ABB RobotStudio station: Romantici.rsstn

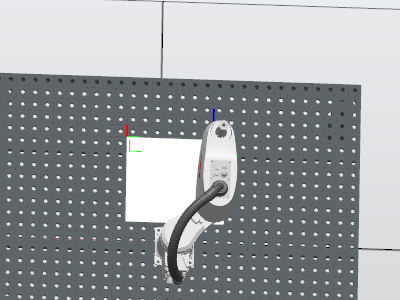
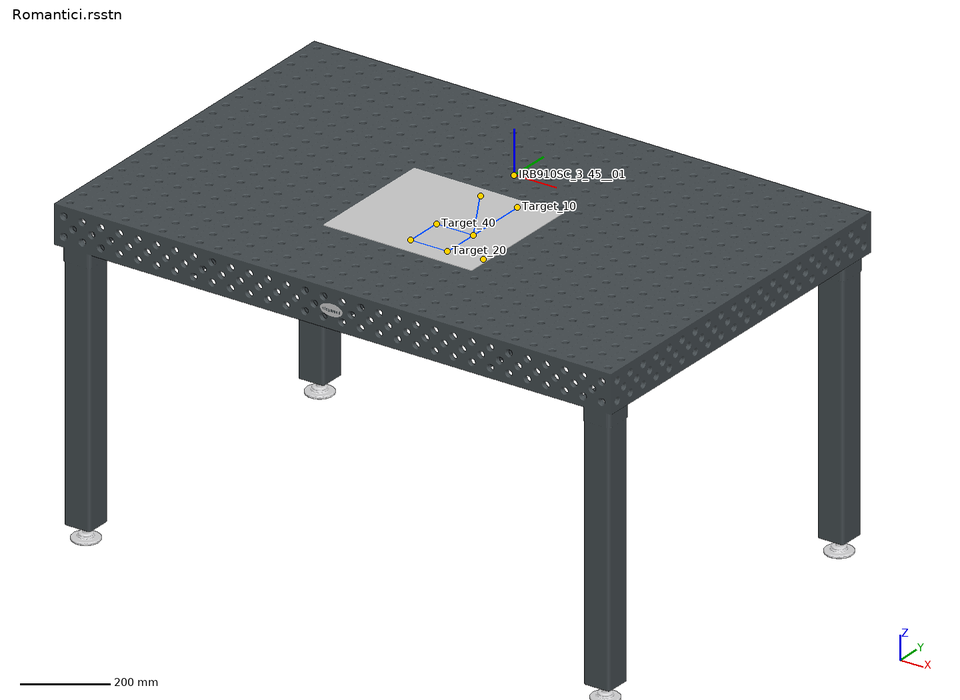
[picture v1: parts stored in the station drawn from their meshes, with robot base, taught points and paths (robot models come from the ABB library and are not in the file)]
Station Solution_1_Tutorial (saved by RobotStudio 22.3.10190.2)
Controller Controller3, task T_ROB1: task frame (RAPID world) sits at (0, 200, 830) mm, rotated rx 0 ry 0 rz -90 deg in the station
Controller Controller3
  mechanical unit ROB_1: IRB910SC_3_45__01, 4 joints, base frame (0, 0, 0) mm
Layout (positions relative to the parent item):
  - table [part] at (-200, -500, 830) mm
  - siegmund_1500_1000 [part], size 1500 x 1010.3 x 830 mm
  - IRB910SC_3_45__01 [mechanism, from Robots\IRB910SC_3_45__01.rslib] at (0, 200, 830) mm, rotated rx 0 ry 0 rz -90 deg; joint values [-2.1543, 2.1819, -0.0556, 0.0276] (rad or m)
  - PencilHolder [mechanism] at (-160, 60.29, 994.64) mm, rotated rx 180 ry 0 rz -90 deg
      TCP PencilHolder at (-72.46, -108.4, 17) mm, rotated rx 90 ry 0 rz 0 deg
      links: Assembly3
  - PAPER [part] at (-200, -250, 830) mm, size 400 x 350 x 2 mm
  - Rámec_1 [frame] at (0, 30, 162.64) mm, rotated rx 90 ry 0 rz -90 deg
Attachment: PencilHolder is attached to IRB910SC_3_45__01 / Link4
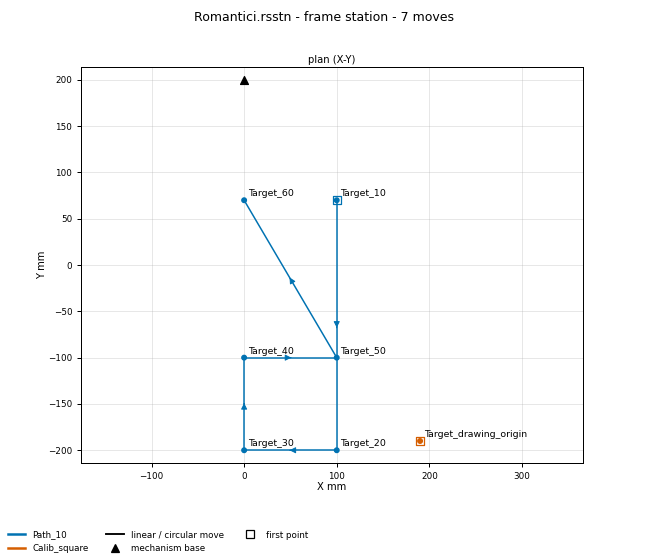
[picture p0: tool path of Romantici.rsstn in frame station, 7 of 7 moves have a stored position in this frame; points joined in program order, loops and branches not executed]
Targets, tools, work objects and paths stored in the station, written as RAPID:
! task T_ROB1
MODULE Module1
  PROC main()
  ENDPROC
ENDMODULE

! task T_ROB2
MODULE Module1
  PROC main()
  ENDPROC
ENDMODULE

! task T_ROB1
MODULE CalibData
  PERS tooldata PencilHolder:=[TRUE,[[0,30,162.643],[1,0,0,0]],[1,[0,0,1],[1,0,0,0],0,0,0]];
  PERS tooldata Pen_TCP:=[TRUE,[[110,0,140],[0.707106781,0,0.707106781,0]],[1,[10.7435139,0,140],[1,0,0,0],0,0,0]];
  TASK PERS wobjdata PAPER:=[FALSE,TRUE,"",[[100,200,0],[0,1,0,0]],[[0,0,0],[1,0,0,0]]];
ENDMODULE

! task T_ROB1
MODULE Module1
  CONST robtarget Target_10:=[[30,100,0],[1,0,0,0],[0,0,0,0],[9E+09,9E+09,9E+09,9E+09,9E+09,9E+09]];
  CONST robtarget Target_20:=[[300,100,0],[1,0,0,0],[0,0,0,0],[9E+09,9E+09,9E+09,9E+09,9E+09,9E+09]];
  CONST robtarget Target_30:=[[300,200,0],[1,0,0,0],[0,0,0,0],[9E+09,9E+09,9E+09,9E+09,9E+09,9E+09]];
  CONST robtarget Target_40:=[[200,200,0],[1,0,0,0],[0,0,0,0],[9E+09,9E+09,9E+09,9E+09,9E+09,9E+09]];
  CONST robtarget Target_50:=[[200,100,0],[1,0,0,0],[0,0,0,0],[9E+09,9E+09,9E+09,9E+09,9E+09,9E+09]];
  CONST robtarget Target_60:=[[30,200,0],[1,0,0,0],[0,0,0,0],[9E+09,9E+09,9E+09,9E+09,9E+09,9E+09]];
  CONST robtarget Target_corner:=[[350,0,-2],[1,0,0,0],[0,0,0,0],[9E+09,9E+09,9E+09,9E+09,9E+09,9E+09]];
  CONST robtarget Target_drawing_origin:=[[290,10,-2],[1,0,0,0],[0,0,0,0],[9E+09,9E+09,9E+09,9E+09,9E+09,9E+09]];
  CONST robtarget Target_opposite_corner:=[[100,390,-2],[1,0,0,0],[0,0,0,0],[9E+09,9E+09,9E+09,9E+09,9E+09,9E+09]];
  PROC Path_10()
    MoveL Target_10,v1000,z0,PencilHolder\WObj:=PAPER;
    MoveL Target_20,v1000,z0,PencilHolder\WObj:=PAPER;
    MoveL Target_30,v1000,z0,PencilHolder\WObj:=PAPER;
    MoveL Target_40,v1000,z0,PencilHolder\WObj:=PAPER;
    MoveL Target_50,v1000,z0,PencilHolder\WObj:=PAPER;
    MoveL Target_60,v1000,z0,PencilHolder\WObj:=PAPER;
  ENDPROC
  PROC main()
  ENDPROC
  PROC Calib_square()
    MoveJ Target_drawing_origin,v1000,z100,PencilHolder\WObj:=PAPER;
  ENDPROC
ENDMODULE

